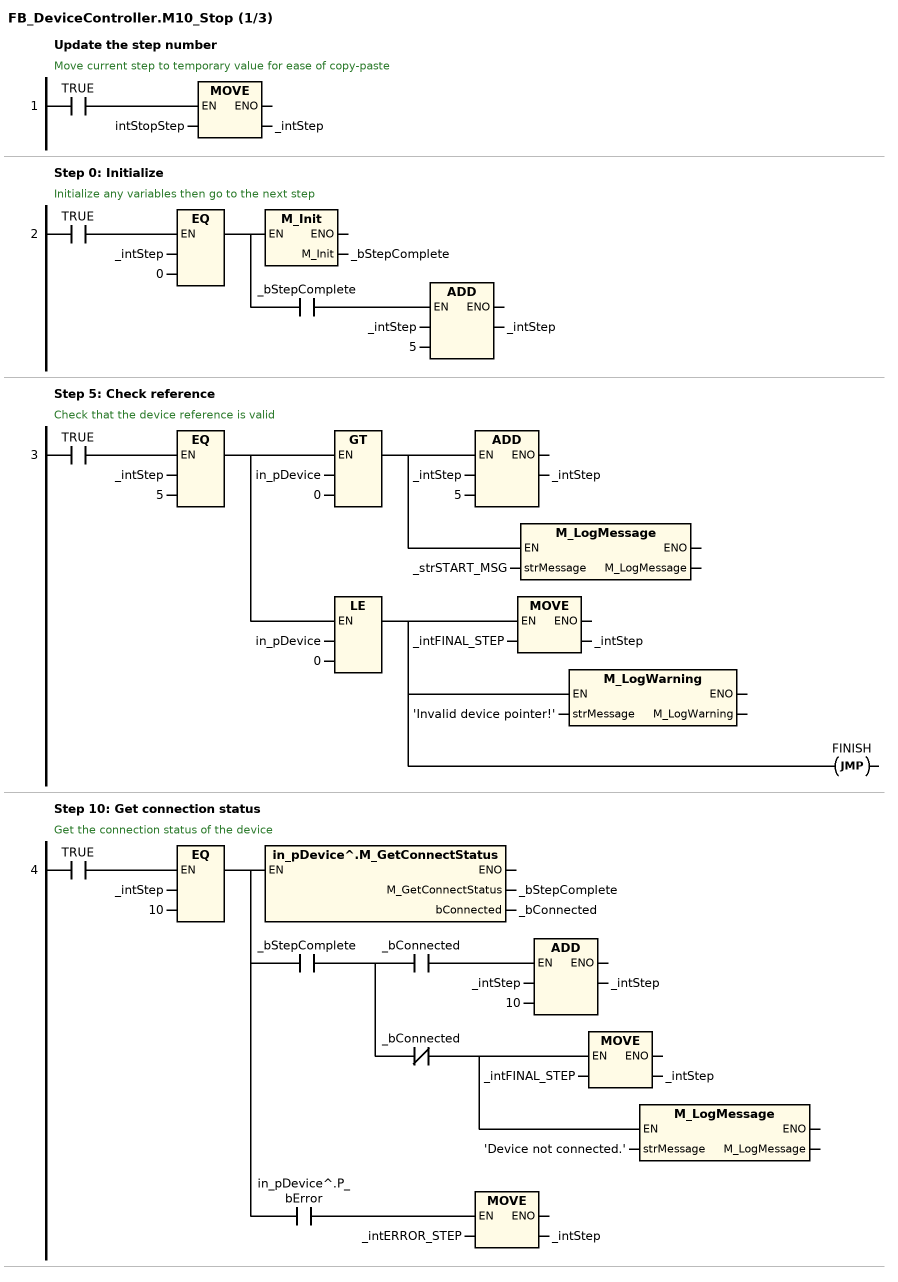
// NETWORK 1: Update the step number
// Move current step to temporary value for ease of copy-paste
_intStep := intStopStep;

// NETWORK 2: Step 0: Initialize
// Initialize any variables then go to the next step
_w1 := _intStep = 0;
IF _w1 THEN _bStepComplete := M_Init(); END_IF
IF _w1 AND _bStepComplete THEN _intStep := _intStep + 5; END_IF

// NETWORK 3: Step 5: Check reference
// Check that the device reference is valid
_w2 := _intStep = 5;
_w3 := _w2 AND in_pDevice > 0;
IF _w3 THEN _intStep := _intStep + 5; END_IF
IF _w3 THEN M_LogMessage(strMessage := _strSTART_MSG); END_IF
_w4 := _w2 AND in_pDevice <= 0;
IF _w4 THEN _intStep := _intFINAL_STEP; END_IF
IF _w4 THEN M_LogWarning(strMessage := 'Invalid device pointer!'); END_IF
IF _w4 THEN JMP FINISH; END_IF

// NETWORK 4: Step 10: Get connection status
// Get the connection status of the device
_w5 := _intStep = 10;
IF _w5 THEN _bStepComplete := in_pDevice^.M_GetConnectStatus(bConnected => _bConnected); END_IF
_w6 := _w5 AND _bStepComplete;
IF _w6 AND _bConnected THEN _intStep := _intStep + 10; END_IF
_w7 := _w6 AND NOT _bConnected;
IF _w7 THEN _intStep := _intFINAL_STEP; END_IF
IF _w7 THEN M_LogMessage(strMessage := 'Device not connected.'); END_IF
IF _w5 AND in_pDevice^.P_bError THEN _intStep := _intERROR_STEP; END_IF

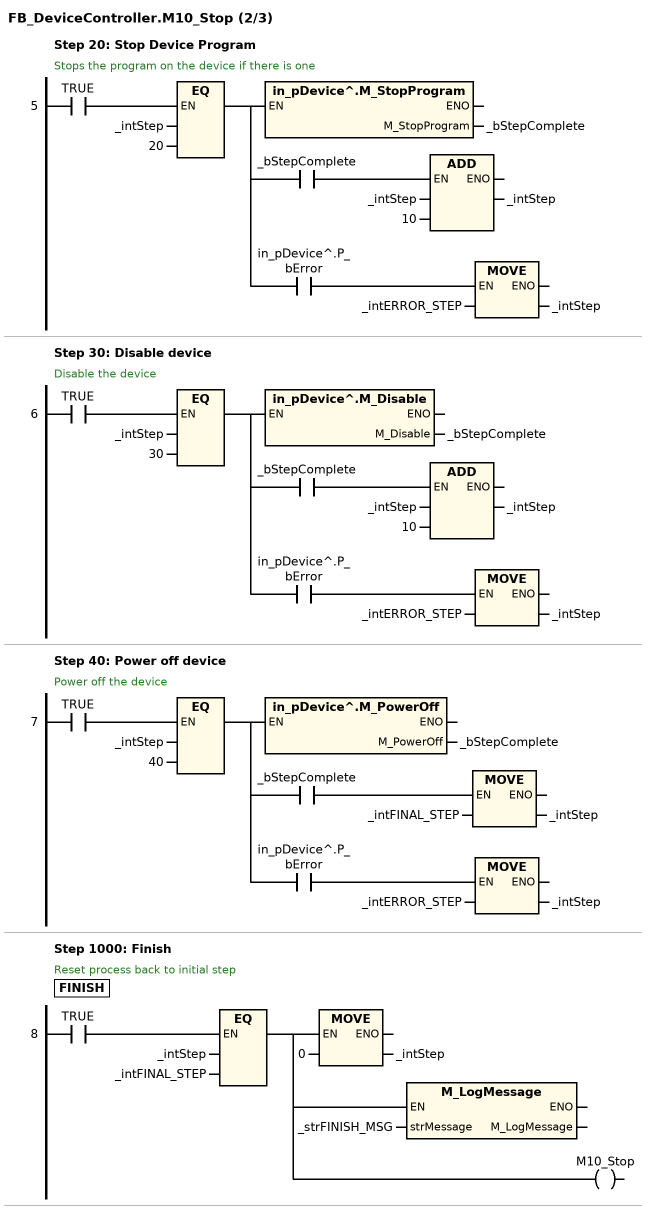
// NETWORK 5: Step 20: Stop Device Program
// Stops the program on the device if there is one
_w8 := _intStep = 20;
IF _w8 THEN _bStepComplete := in_pDevice^.M_StopProgram(); END_IF
IF _w8 AND _bStepComplete THEN _intStep := _intStep + 10; END_IF
IF _w8 AND in_pDevice^.P_bError THEN _intStep := _intERROR_STEP; END_IF

// NETWORK 6: Step 30: Disable device
// Disable the device
_w9 := _intStep = 30;
IF _w9 THEN _bStepComplete := in_pDevice^.M_Disable(); END_IF
IF _w9 AND _bStepComplete THEN _intStep := _intStep + 10; END_IF
IF _w9 AND in_pDevice^.P_bError THEN _intStep := _intERROR_STEP; END_IF

// NETWORK 7: Step 40: Power off device
// Power off the device
_w10 := _intStep = 40;
IF _w10 THEN _bStepComplete := in_pDevice^.M_PowerOff(); END_IF
IF _w10 AND _bStepComplete THEN _intStep := _intFINAL_STEP; END_IF
IF _w10 AND in_pDevice^.P_bError THEN _intStep := _intERROR_STEP; END_IF

// NETWORK 8: Step 1000: Finish
// Reset process back to initial step
FINISH:
_w11 := _intStep = _intFINAL_STEP;
IF _w11 THEN _intStep := 0; END_IF
IF _w11 THEN M_LogMessage(strMessage := _strFINISH_MSG); END_IF
M10_Stop := _w11;

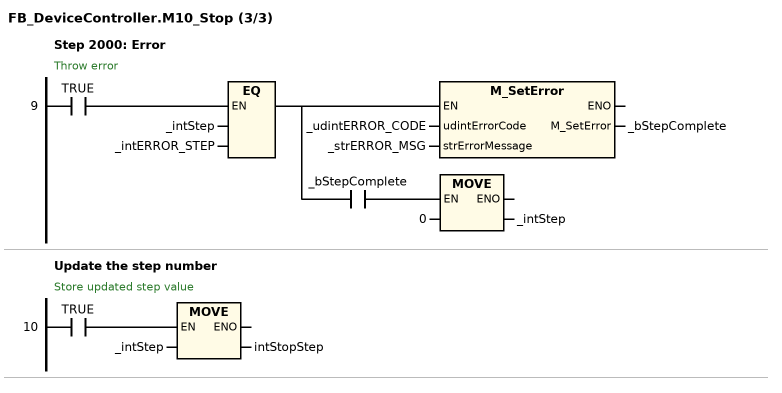
// NETWORK 9: Step 2000: Error
// Throw error
_w12 := _intStep = _intERROR_STEP;
IF _w12 THEN
    _bStepComplete := M_SetError(udintErrorCode := _udintERROR_CODE, strErrorMessage := _strERROR_MSG);
END_IF
IF _w12 AND _bStepComplete THEN _intStep := 0; END_IF

// NETWORK 10: Update the step number
// Store updated step value
intStopStep := _intStep;
END_METHOD

(* Connects, resets, and powers on the device. *)
METHOD M20_Reset : BOOL
VAR CONSTANT
	_intFINAL_STEP : INT := 1000;
	_intERROR_STEP : INT := 2000;
	_udintERROR_CODE: UDINT := E_DeviceControllerError.ResetError;
	_strERROR_MSG: T_MaxString := 'Error while trying to reset device!';
	_strSTART_MSG: T_MaxString := 'Resetting device';
	_strFINISH_MSG: T_MaxString := 'Device reset';
END_VAR
VAR
	_bStepComplete: BOOL;
	_intStep: INT;
END_VAR
VAR_INST // added by the converter: edge detectors and wires of the graphical bodies
    _w1, _w2, _w3, _w4, _w5, _w6, _w7, _w8, _w9 : BOOL;
END_VAR
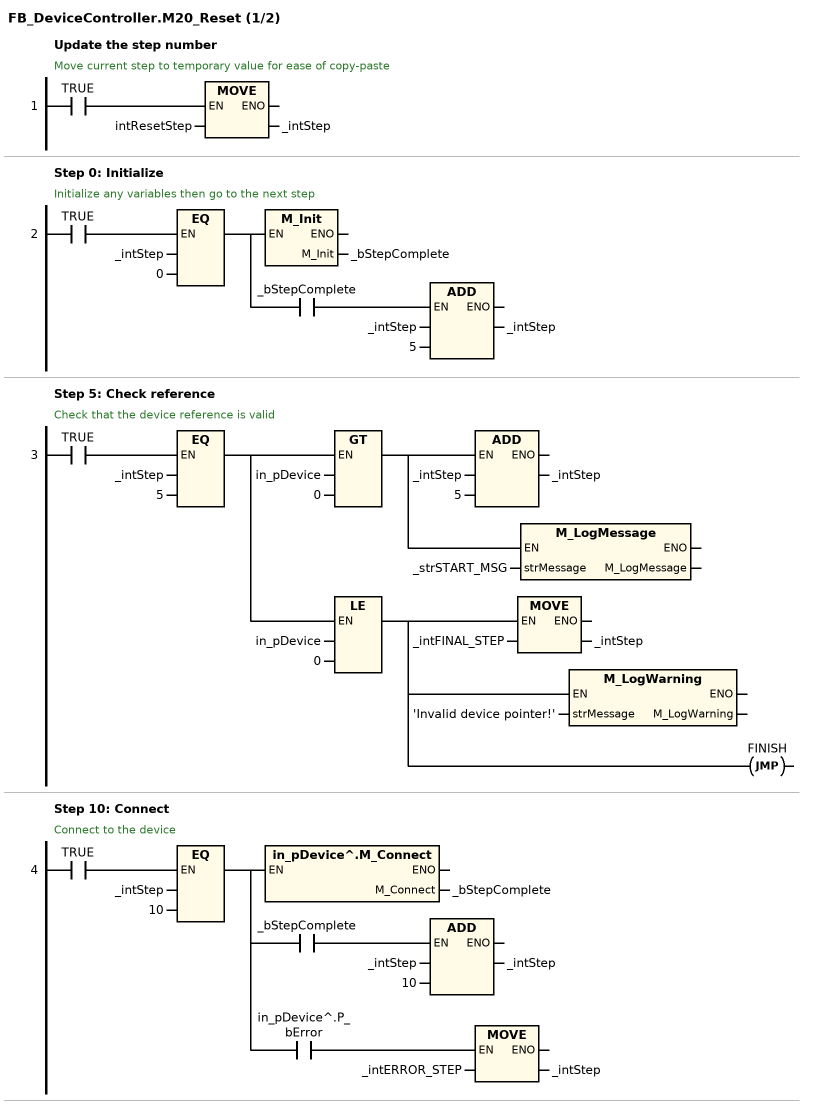
// NETWORK 1: Update the step number
// Move current step to temporary value for ease of copy-paste
_intStep := intResetStep;

// NETWORK 2: Step 0: Initialize
// Initialize any variables then go to the next step
_w1 := _intStep = 0;
IF _w1 THEN _bStepComplete := M_Init(); END_IF
IF _w1 AND _bStepComplete THEN _intStep := _intStep + 5; END_IF

// NETWORK 3: Step 5: Check reference
// Check that the device reference is valid
_w2 := _intStep = 5;
_w3 := _w2 AND in_pDevice > 0;
IF _w3 THEN _intStep := _intStep + 5; END_IF
IF _w3 THEN M_LogMessage(strMessage := _strSTART_MSG); END_IF
_w4 := _w2 AND in_pDevice <= 0;
IF _w4 THEN _intStep := _intFINAL_STEP; END_IF
IF _w4 THEN M_LogWarning(strMessage := 'Invalid device pointer!'); END_IF
IF _w4 THEN JMP FINISH; END_IF

// NETWORK 4: Step 10: Connect
// Connect to the device
_w5 := _intStep = 10;
IF _w5 THEN _bStepComplete := in_pDevice^.M_Connect(); END_IF
IF _w5 AND _bStepComplete THEN _intStep := _intStep + 10; END_IF
IF _w5 AND in_pDevice^.P_bError THEN _intStep := _intERROR_STEP; END_IF

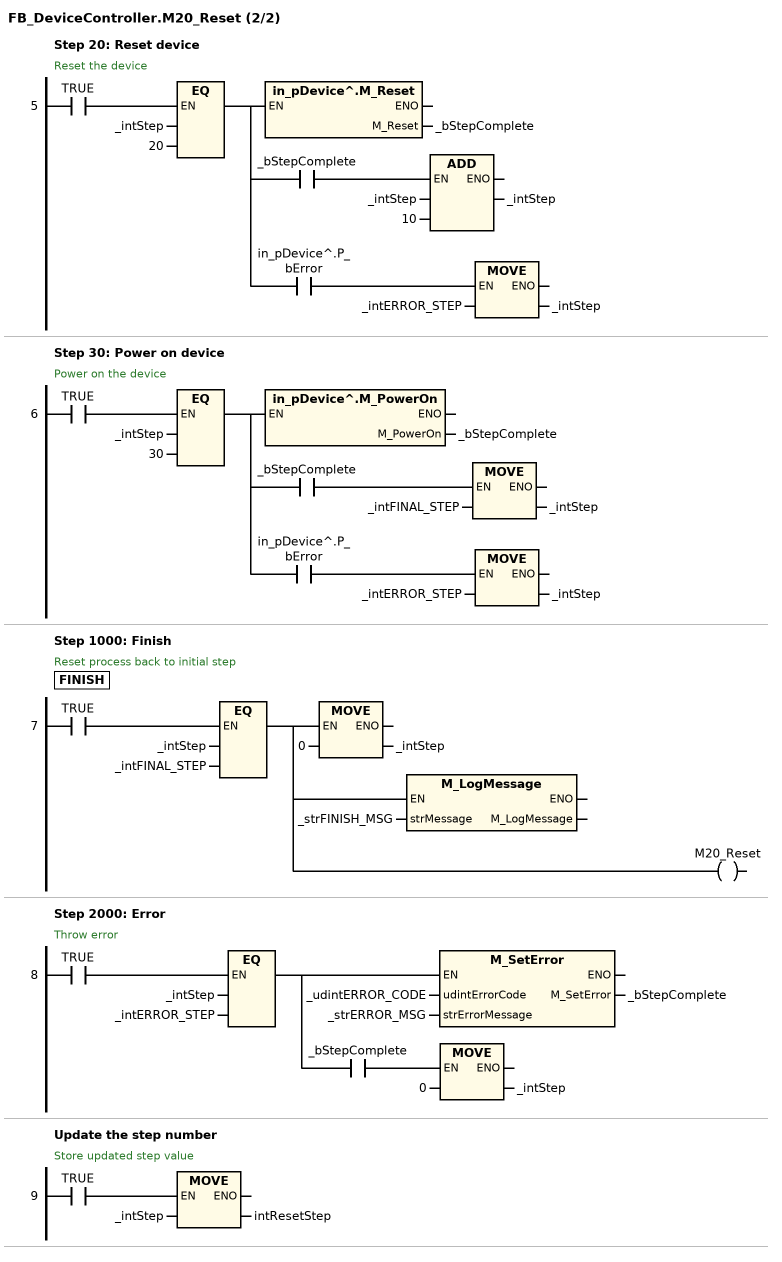
// NETWORK 5: Step 20: Reset device
// Reset the device
_w6 := _intStep = 20;
IF _w6 THEN _bStepComplete := in_pDevice^.M_Reset(); END_IF
IF _w6 AND _bStepComplete THEN _intStep := _intStep + 10; END_IF
IF _w6 AND in_pDevice^.P_bError THEN _intStep := _intERROR_STEP; END_IF

// NETWORK 6: Step 30: Power on device
// Power on the device
_w7 := _intStep = 30;
IF _w7 THEN _bStepComplete := in_pDevice^.M_PowerOn(); END_IF
IF _w7 AND _bStepComplete THEN _intStep := _intFINAL_STEP; END_IF
IF _w7 AND in_pDevice^.P_bError THEN _intStep := _intERROR_STEP; END_IF

// NETWORK 7: Step 1000: Finish
// Reset process back to initial step
FINISH:
_w8 := _intStep = _intFINAL_STEP;
IF _w8 THEN _intStep := 0; END_IF
IF _w8 THEN M_LogMessage(strMessage := _strFINISH_MSG); END_IF
M20_Reset := _w8;

// NETWORK 8: Step 2000: Error
// Throw error
_w9 := _intStep = _intERROR_STEP;
IF _w9 THEN
    _bStepComplete := M_SetError(udintErrorCode := _udintERROR_CODE, strErrorMessage := _strERROR_MSG);
END_IF
IF _w9 AND _bStepComplete THEN _intStep := 0; END_IF

// NETWORK 9: Update the step number
// Store updated step value
intResetStep := _intStep;
END_METHOD

(* Loads program and starts device then returns TRUE. *)
METHOD M30_Start : BOOL
VAR CONSTANT
	_udintERROR_CODE: UDINT := E_DeviceControllerError.StartError;
	_strERROR_MSG: T_MaxString := 'Error while trying to start device!';
	_intFINAL_STEP : INT := 1000;
	_intERROR_STEP : INT := 2000;
	_strSTART_MSG: T_MaxString := 'Starting device';
	_strFINISH_MSG: T_MaxString := 'Device started';
END_VAR
VAR
	_bStepComplete: BOOL;
	_intStep: INT;
END_VAR
VAR_INST // added by the converter: edge detectors and wires of the graphical bodies
    _w1, _w2, _w3, _w4, _w5, _w6, _w7, _w8, _w9 : BOOL;
END_VAR
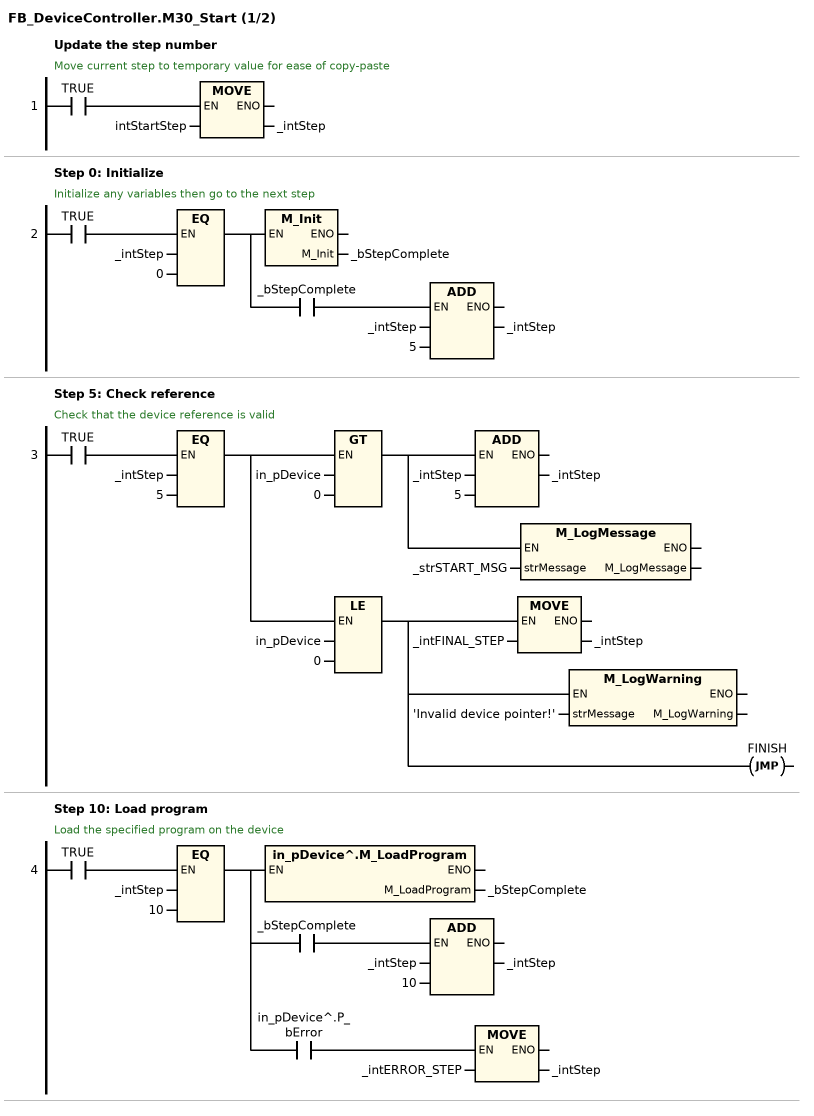
// NETWORK 1: Update the step number
// Move current step to temporary value for ease of copy-paste
_intStep := intStartStep;

// NETWORK 2: Step 0: Initialize
// Initialize any variables then go to the next step
_w1 := _intStep = 0;
IF _w1 THEN _bStepComplete := M_Init(); END_IF
IF _w1 AND _bStepComplete THEN _intStep := _intStep + 5; END_IF

// NETWORK 3: Step 5: Check reference
// Check that the device reference is valid
_w2 := _intStep = 5;
_w3 := _w2 AND in_pDevice > 0;
IF _w3 THEN _intStep := _intStep + 5; END_IF
IF _w3 THEN M_LogMessage(strMessage := _strSTART_MSG); END_IF
_w4 := _w2 AND in_pDevice <= 0;
IF _w4 THEN _intStep := _intFINAL_STEP; END_IF
IF _w4 THEN M_LogWarning(strMessage := 'Invalid device pointer!'); END_IF
IF _w4 THEN JMP FINISH; END_IF

// NETWORK 4: Step 10: Load program
// Load the specified program on the device
_w5 := _intStep = 10;
IF _w5 THEN _bStepComplete := in_pDevice^.M_LoadProgram(); END_IF
IF _w5 AND _bStepComplete THEN _intStep := _intStep + 10; END_IF
IF _w5 AND in_pDevice^.P_bError THEN _intStep := _intERROR_STEP; END_IF

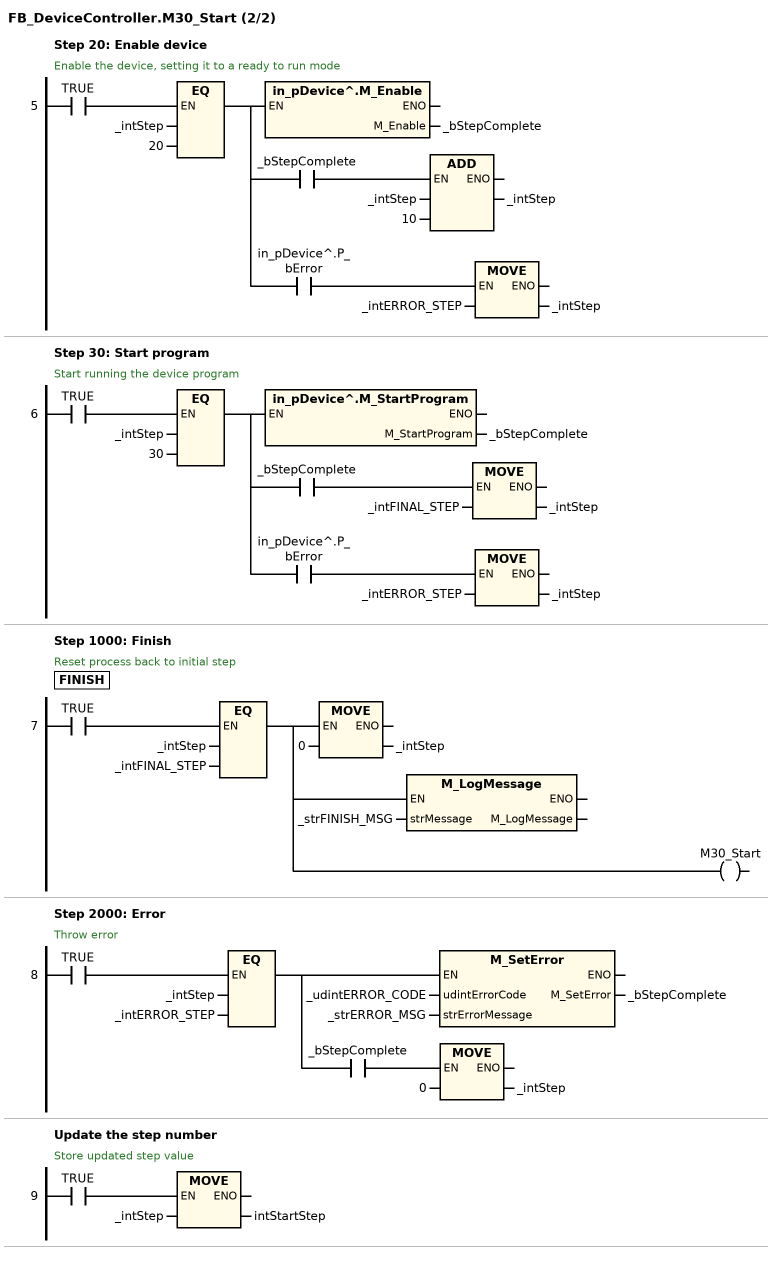
// NETWORK 5: Step 20: Enable device
// Enable the device, setting it to a ready to run mode
_w6 := _intStep = 20;
IF _w6 THEN _bStepComplete := in_pDevice^.M_Enable(); END_IF
IF _w6 AND _bStepComplete THEN _intStep := _intStep + 10; END_IF
IF _w6 AND in_pDevice^.P_bError THEN _intStep := _intERROR_STEP; END_IF

// NETWORK 6: Step 30: Start program
// Start running the device program
_w7 := _intStep = 30;
IF _w7 THEN _bStepComplete := in_pDevice^.M_StartProgram(); END_IF
IF _w7 AND _bStepComplete THEN _intStep := _intFINAL_STEP; END_IF
IF _w7 AND in_pDevice^.P_bError THEN _intStep := _intERROR_STEP; END_IF

// NETWORK 7: Step 1000: Finish
// Reset process back to initial step
FINISH:
_w8 := _intStep = _intFINAL_STEP;
IF _w8 THEN _intStep := 0; END_IF
IF _w8 THEN M_LogMessage(strMessage := _strFINISH_MSG); END_IF
M30_Start := _w8;

// NETWORK 8: Step 2000: Error
// Throw error
_w9 := _intStep = _intERROR_STEP;
IF _w9 THEN
    _bStepComplete := M_SetError(udintErrorCode := _udintERROR_CODE, strErrorMessage := _strERROR_MSG);
END_IF
IF _w9 AND _bStepComplete THEN _intStep := 0; END_IF

// NETWORK 9: Update the step number
// Store updated step value
intStartStep := _intStep;
END_METHOD

(* Stops and disables the device then returns TRUE when done. *)
METHOD M32_Complete : BOOL
VAR CONSTANT
	_udintERROR_CODE: UDINT := E_DeviceControllerError.CompleteError;
	_strERROR_MSG: T_MaxString := 'Error while trying to complete device!';
	_intFINAL_STEP : INT := 1000;
	_intERROR_STEP : INT := 2000;
	_strSTART_MSG: T_MaxString := 'Completing device';
	_strFINISH_MSG: T_MaxString := 'Device completed';
END_VAR
VAR
	_bStepComplete: BOOL;
	_intStep: INT;
END_VAR
VAR_INST // added by the converter: edge detectors and wires of the graphical bodies
    _w1, _w2, _w3, _w4, _w5, _w6, _w7, _w8 : BOOL;
END_VAR
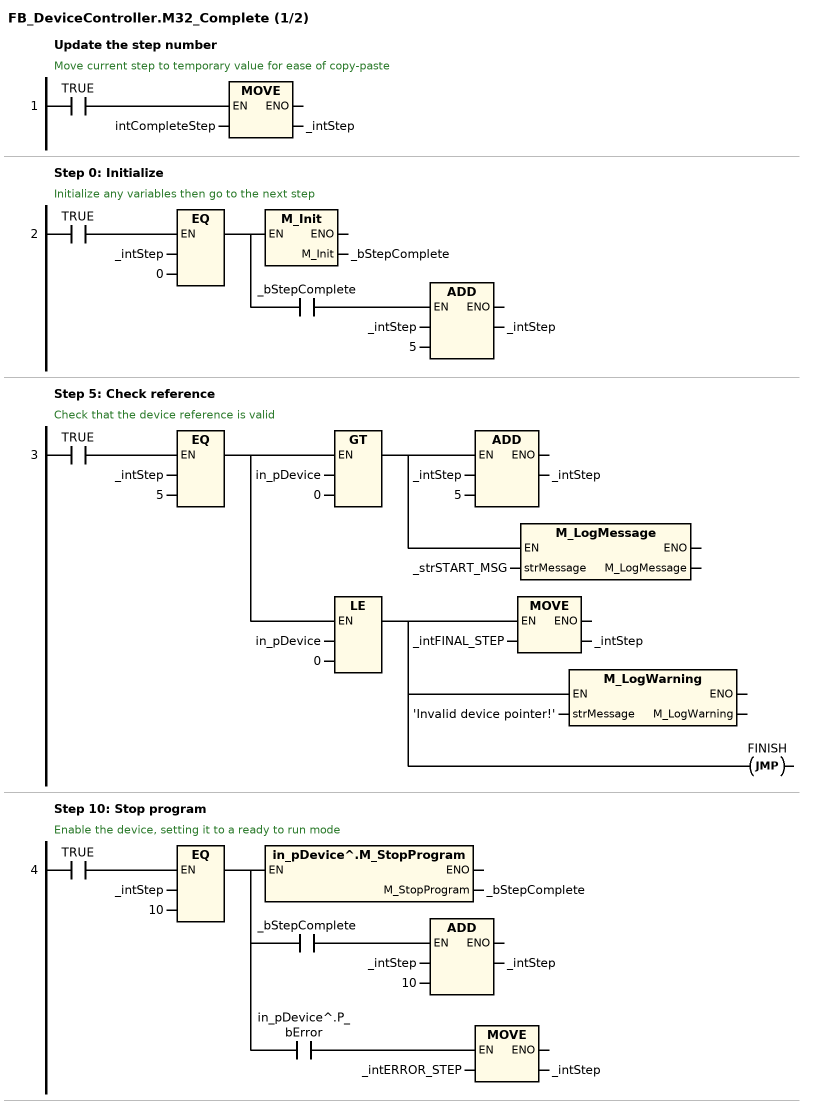
// NETWORK 1: Update the step number
// Move current step to temporary value for ease of copy-paste
_intStep := intCompleteStep;

// NETWORK 2: Step 0: Initialize
// Initialize any variables then go to the next step
_w1 := _intStep = 0;
IF _w1 THEN _bStepComplete := M_Init(); END_IF
IF _w1 AND _bStepComplete THEN _intStep := _intStep + 5; END_IF

// NETWORK 3: Step 5: Check reference
// Check that the device reference is valid
_w2 := _intStep = 5;
_w3 := _w2 AND in_pDevice > 0;
IF _w3 THEN _intStep := _intStep + 5; END_IF
IF _w3 THEN M_LogMessage(strMessage := _strSTART_MSG); END_IF
_w4 := _w2 AND in_pDevice <= 0;
IF _w4 THEN _intStep := _intFINAL_STEP; END_IF
IF _w4 THEN M_LogWarning(strMessage := 'Invalid device pointer!'); END_IF
IF _w4 THEN JMP FINISH; END_IF

// NETWORK 4: Step 10: Stop program
// Enable the device, setting it to a ready to run mode
_w5 := _intStep = 10;
IF _w5 THEN _bStepComplete := in_pDevice^.M_StopProgram(); END_IF
IF _w5 AND _bStepComplete THEN _intStep := _intStep + 10; END_IF
IF _w5 AND in_pDevice^.P_bError THEN _intStep := _intERROR_STEP; END_IF

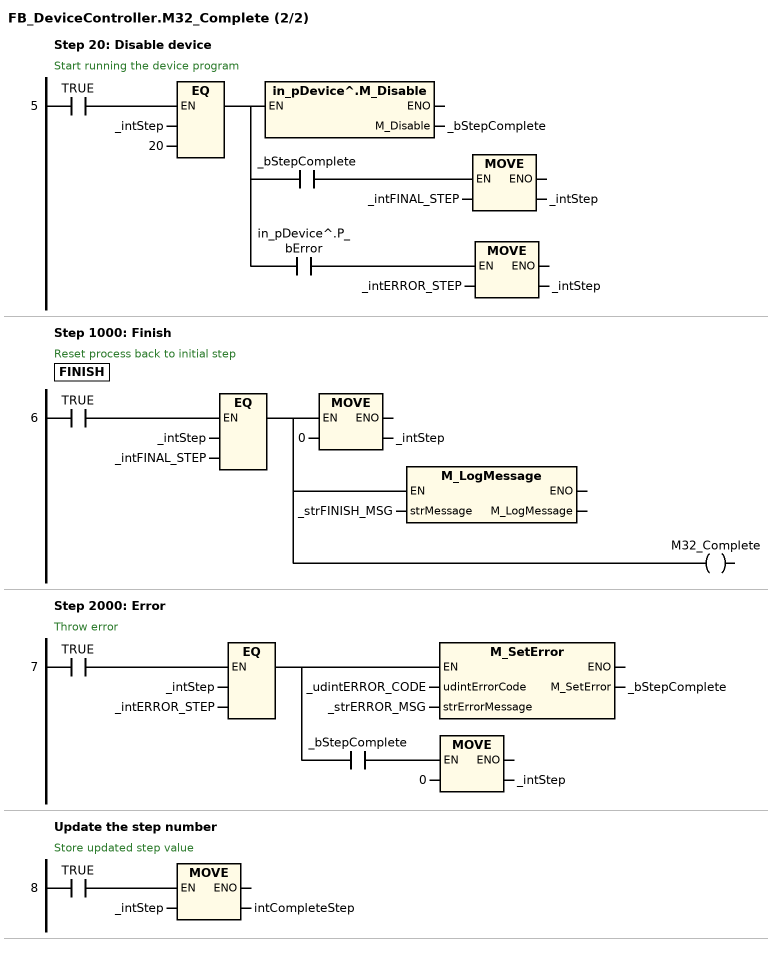
// NETWORK 5: Step 20: Disable device
// Start running the device program
_w6 := _intStep = 20;
IF _w6 THEN _bStepComplete := in_pDevice^.M_Disable(); END_IF
IF _w6 AND _bStepComplete THEN _intStep := _intFINAL_STEP; END_IF
IF _w6 AND in_pDevice^.P_bError THEN _intStep := _intERROR_STEP; END_IF

// NETWORK 6: Step 1000: Finish
// Reset process back to initial step
FINISH:
_w7 := _intStep = _intFINAL_STEP;
IF _w7 THEN _intStep := 0; END_IF
IF _w7 THEN M_LogMessage(strMessage := _strFINISH_MSG); END_IF
M32_Complete := _w7;

// NETWORK 7: Step 2000: Error
// Throw error
_w8 := _intStep = _intERROR_STEP;
IF _w8 THEN
    _bStepComplete := M_SetError(udintErrorCode := _udintERROR_CODE, strErrorMessage := _strERROR_MSG);
END_IF
IF _w8 AND _bStepComplete THEN _intStep := 0; END_IF

// NETWORK 8: Update the step number
// Store updated step value
intCompleteStep := _intStep;
END_METHOD

(* Pauses the device then returns TRUE. *)
METHOD M40_Hold : BOOL
VAR CONSTANT
	_udintERROR_CODE: UDINT := E_DeviceControllerError.HoldError;
	_strERROR_MSG: T_MaxString := 'Error while trying to hold device!';
	_intFINAL_STEP : INT := 1000;
	_intERROR_STEP : INT := 2000;
	_strSTART_MSG: T_MaxString := 'Holding device';
	_strFINISH_MSG: T_MaxString := 'Device held';
END_VAR
VAR
	_bStepComplete: BOOL;
	_intStep: INT;
END_VAR
VAR_INST // added by the converter: edge detectors and wires of the graphical bodies
    _w1, _w2, _w3, _w4, _w5, _w6, _w7 : BOOL;
END_VAR
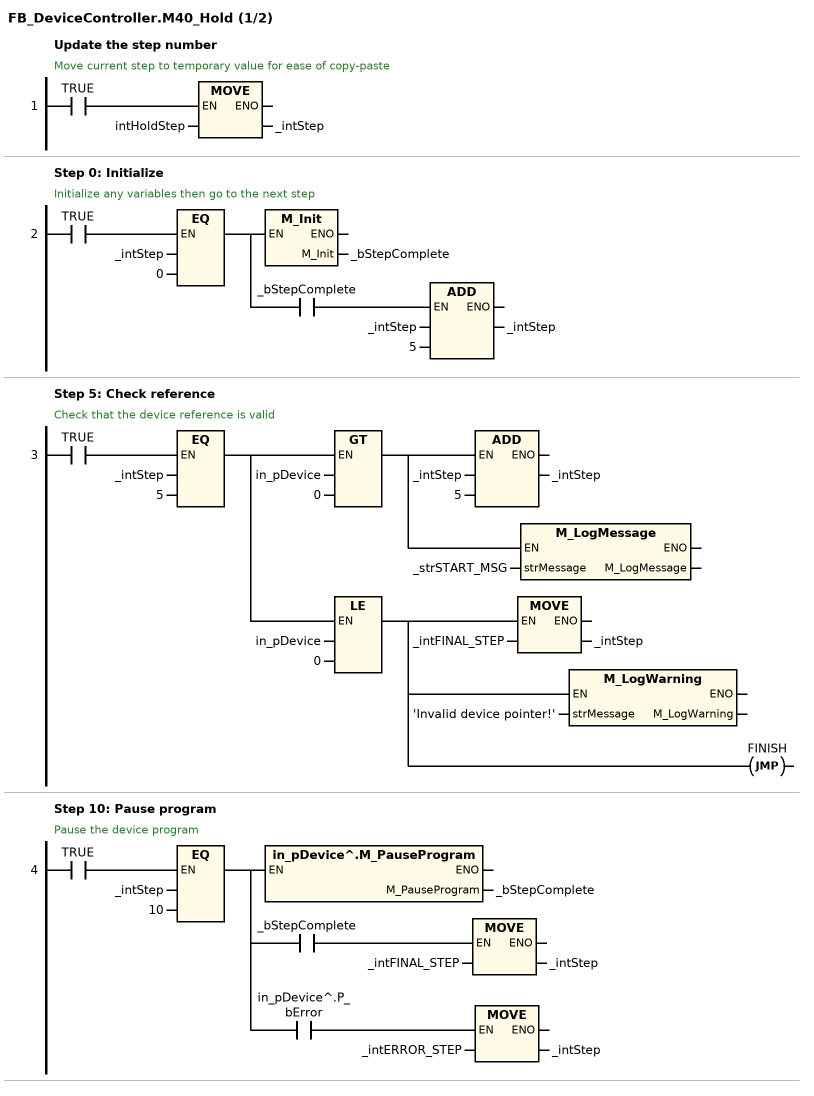
// NETWORK 1: Update the step number
// Move current step to temporary value for ease of copy-paste
_intStep := intHoldStep;

// NETWORK 2: Step 0: Initialize
// Initialize any variables then go to the next step
_w1 := _intStep = 0;
IF _w1 THEN _bStepComplete := M_Init(); END_IF
IF _w1 AND _bStepComplete THEN _intStep := _intStep + 5; END_IF

// NETWORK 3: Step 5: Check reference
// Check that the device reference is valid
_w2 := _intStep = 5;
_w3 := _w2 AND in_pDevice > 0;
IF _w3 THEN _intStep := _intStep + 5; END_IF
IF _w3 THEN M_LogMessage(strMessage := _strSTART_MSG); END_IF
_w4 := _w2 AND in_pDevice <= 0;
IF _w4 THEN _intStep := _intFINAL_STEP; END_IF
IF _w4 THEN M_LogWarning(strMessage := 'Invalid device pointer!'); END_IF
IF _w4 THEN JMP FINISH; END_IF

// NETWORK 4: Step 10: Pause program
// Pause the device program
_w5 := _intStep = 10;
IF _w5 THEN _bStepComplete := in_pDevice^.M_PauseProgram(); END_IF
IF _w5 AND _bStepComplete THEN _intStep := _intFINAL_STEP; END_IF
IF _w5 AND in_pDevice^.P_bError THEN _intStep := _intERROR_STEP; END_IF

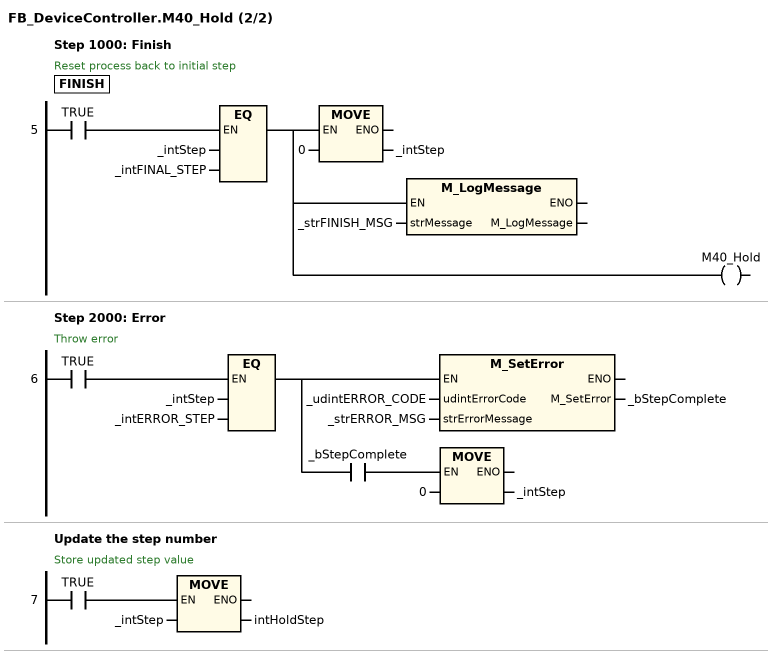
// NETWORK 5: Step 1000: Finish
// Reset process back to initial step
FINISH:
_w6 := _intStep = _intFINAL_STEP;
IF _w6 THEN _intStep := 0; END_IF
IF _w6 THEN M_LogMessage(strMessage := _strFINISH_MSG); END_IF
M40_Hold := _w6;

// NETWORK 6: Step 2000: Error
// Throw error
_w7 := _intStep = _intERROR_STEP;
IF _w7 THEN
    _bStepComplete := M_SetError(udintErrorCode := _udintERROR_CODE, strErrorMessage := _strERROR_MSG);
END_IF
IF _w7 AND _bStepComplete THEN _intStep := 0; END_IF

// NETWORK 7: Update the step number
// Store updated step value
intHoldStep := _intStep;
END_METHOD

(* Unpauses the device then returns TRUE. *)
METHOD M42_Unhold : BOOL
VAR CONSTANT
	_udintERROR_CODE: UDINT := E_DeviceControllerError.UnholdError;
	_strERROR_MSG: T_MaxString := 'Error while trying to unhold device!';
	_intFINAL_STEP : INT := 1000;
	_intERROR_STEP : INT := 2000;
	_strSTART_MSG: T_MaxString := 'Unholding device';
	_strFINISH_MSG: T_MaxString := 'Device unheld';
END_VAR
VAR
	_bStepComplete: BOOL;
	_intStep: INT;
END_VAR
VAR_INST // added by the converter: edge detectors and wires of the graphical bodies
    _w1, _w2, _w3, _w4, _w5, _w6, _w7 : BOOL;
END_VAR
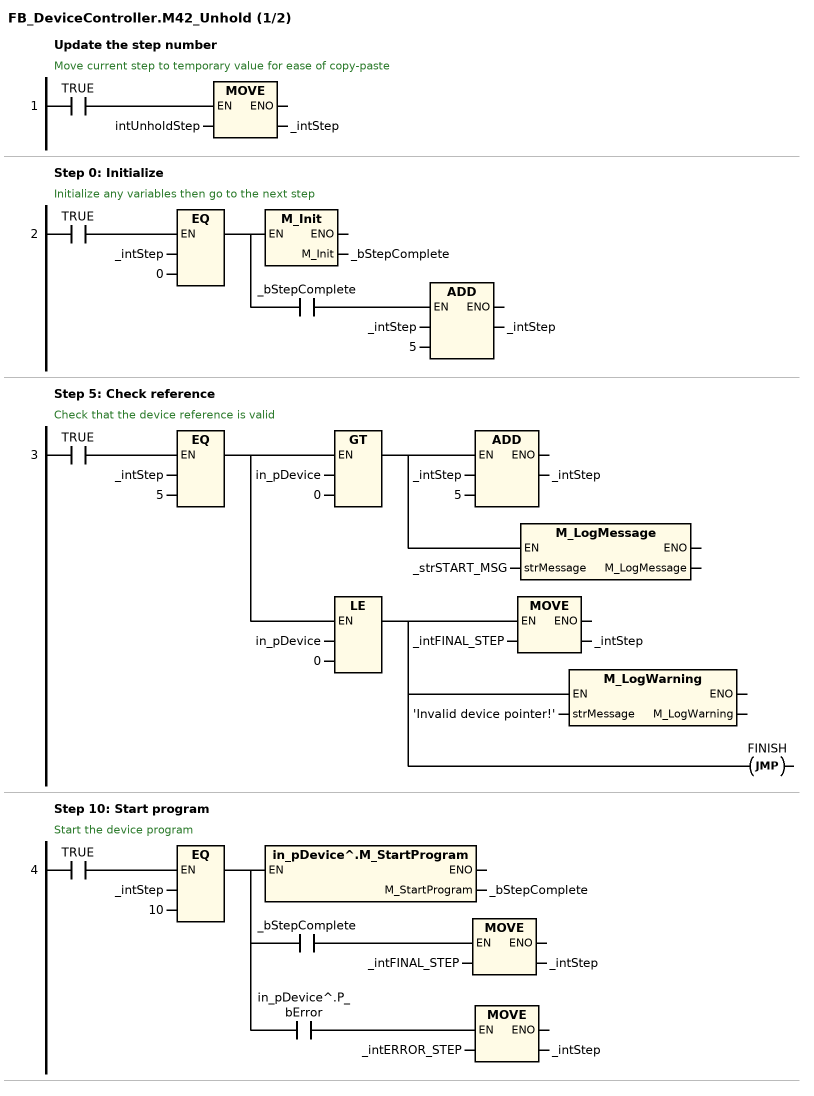
// NETWORK 1: Update the step number
// Move current step to temporary value for ease of copy-paste
_intStep := intUnholdStep;

// NETWORK 2: Step 0: Initialize
// Initialize any variables then go to the next step
_w1 := _intStep = 0;
IF _w1 THEN _bStepComplete := M_Init(); END_IF
IF _w1 AND _bStepComplete THEN _intStep := _intStep + 5; END_IF

// NETWORK 3: Step 5: Check reference
// Check that the device reference is valid
_w2 := _intStep = 5;
_w3 := _w2 AND in_pDevice > 0;
IF _w3 THEN _intStep := _intStep + 5; END_IF
IF _w3 THEN M_LogMessage(strMessage := _strSTART_MSG); END_IF
_w4 := _w2 AND in_pDevice <= 0;
IF _w4 THEN _intStep := _intFINAL_STEP; END_IF
IF _w4 THEN M_LogWarning(strMessage := 'Invalid device pointer!'); END_IF
IF _w4 THEN JMP FINISH; END_IF

// NETWORK 4: Step 10: Start program
// Start the device program
_w5 := _intStep = 10;
IF _w5 THEN _bStepComplete := in_pDevice^.M_StartProgram(); END_IF
IF _w5 AND _bStepComplete THEN _intStep := _intFINAL_STEP; END_IF
IF _w5 AND in_pDevice^.P_bError THEN _intStep := _intERROR_STEP; END_IF

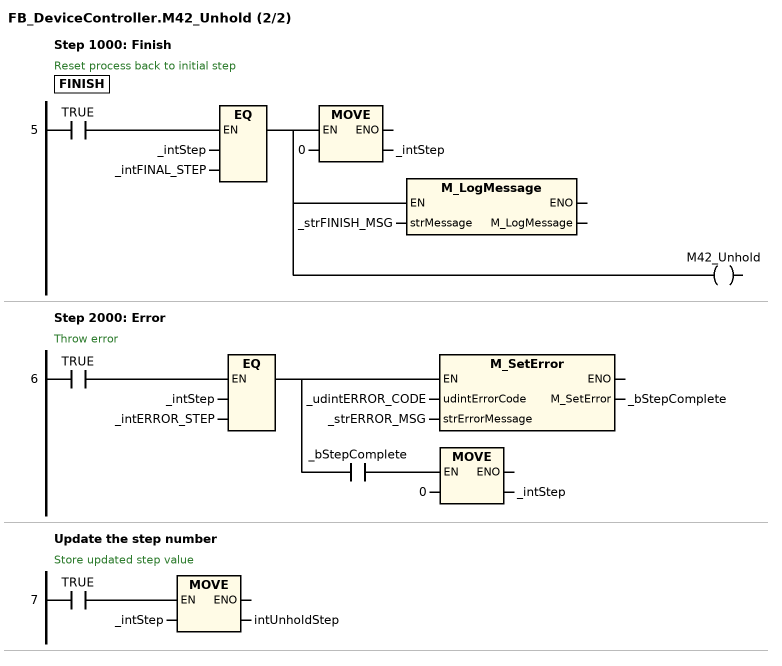
// NETWORK 5: Step 1000: Finish
// Reset process back to initial step
FINISH:
_w6 := _intStep = _intFINAL_STEP;
IF _w6 THEN _intStep := 0; END_IF
IF _w6 THEN M_LogMessage(strMessage := _strFINISH_MSG); END_IF
M42_Unhold := _w6;

// NETWORK 6: Step 2000: Error
// Throw error
_w7 := _intStep = _intERROR_STEP;
IF _w7 THEN
    _bStepComplete := M_SetError(udintErrorCode := _udintERROR_CODE, strErrorMessage := _strERROR_MSG);
END_IF
IF _w7 AND _bStepComplete THEN _intStep := 0; END_IF

// NETWORK 7: Update the step number
// Store updated step value
intUnholdStep := _intStep;
END_METHOD

(* Pauses the device then returns TRUE. *)
METHOD M50_Suspend : BOOL
VAR CONSTANT
	_udintERROR_CODE: UDINT := E_DeviceControllerError.SuspendError;
	_strERROR_MSG: T_MaxString := 'Error while trying to suspend device!';
	_intFINAL_STEP : INT := 1000;
	_intERROR_STEP : INT := 2000;
	_strSTART_MSG: T_MaxString := 'Suspending device';
	_strFINISH_MSG: T_MaxString := 'Device suspended';
END_VAR
VAR
	_bStepComplete: BOOL;
	_intStep: INT;
END_VAR
VAR_INST // added by the converter: edge detectors and wires of the graphical bodies
    _w1, _w2, _w3, _w4, _w5, _w6, _w7 : BOOL;
END_VAR
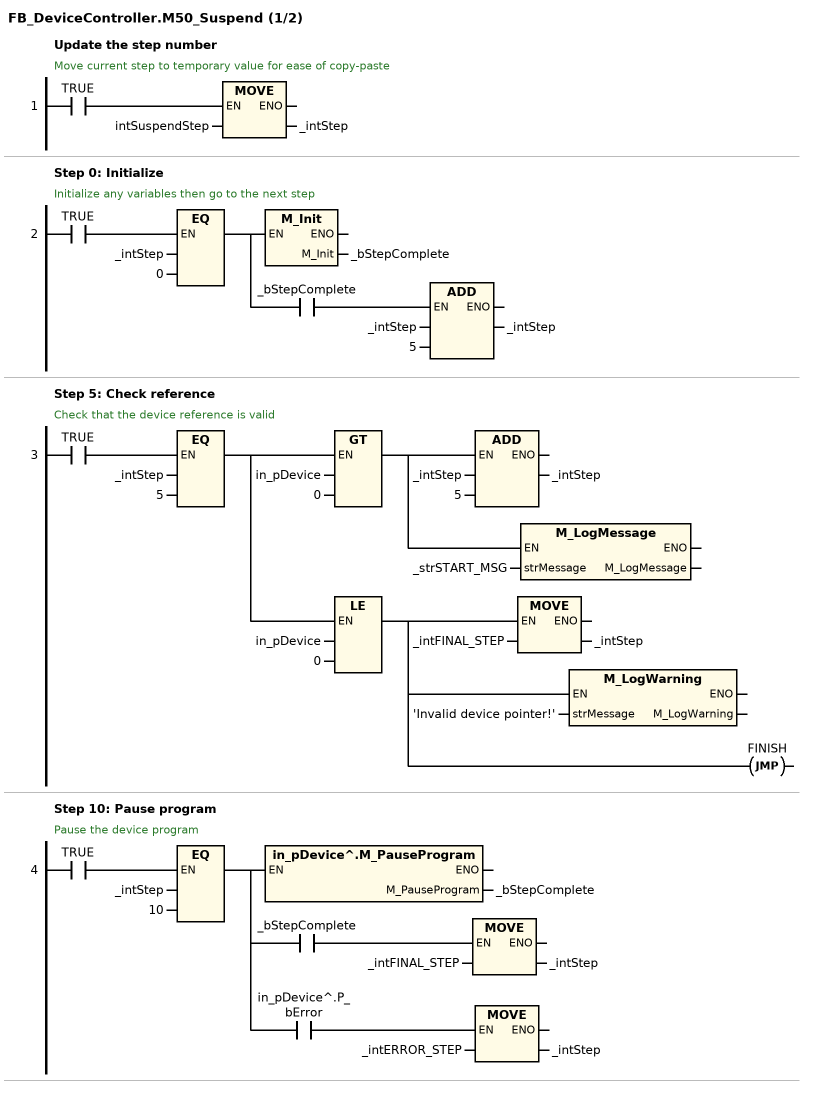
// NETWORK 1: Update the step number
// Move current step to temporary value for ease of copy-paste
_intStep := intSuspendStep;

// NETWORK 2: Step 0: Initialize
// Initialize any variables then go to the next step
_w1 := _intStep = 0;
IF _w1 THEN _bStepComplete := M_Init(); END_IF
IF _w1 AND _bStepComplete THEN _intStep := _intStep + 5; END_IF

// NETWORK 3: Step 5: Check reference
// Check that the device reference is valid
_w2 := _intStep = 5;
_w3 := _w2 AND in_pDevice > 0;
IF _w3 THEN _intStep := _intStep + 5; END_IF
IF _w3 THEN M_LogMessage(strMessage := _strSTART_MSG); END_IF
_w4 := _w2 AND in_pDevice <= 0;
IF _w4 THEN _intStep := _intFINAL_STEP; END_IF
IF _w4 THEN M_LogWarning(strMessage := 'Invalid device pointer!'); END_IF
IF _w4 THEN JMP FINISH; END_IF

// NETWORK 4: Step 10: Pause program
// Pause the device program
_w5 := _intStep = 10;
IF _w5 THEN _bStepComplete := in_pDevice^.M_PauseProgram(); END_IF
IF _w5 AND _bStepComplete THEN _intStep := _intFINAL_STEP; END_IF
IF _w5 AND in_pDevice^.P_bError THEN _intStep := _intERROR_STEP; END_IF

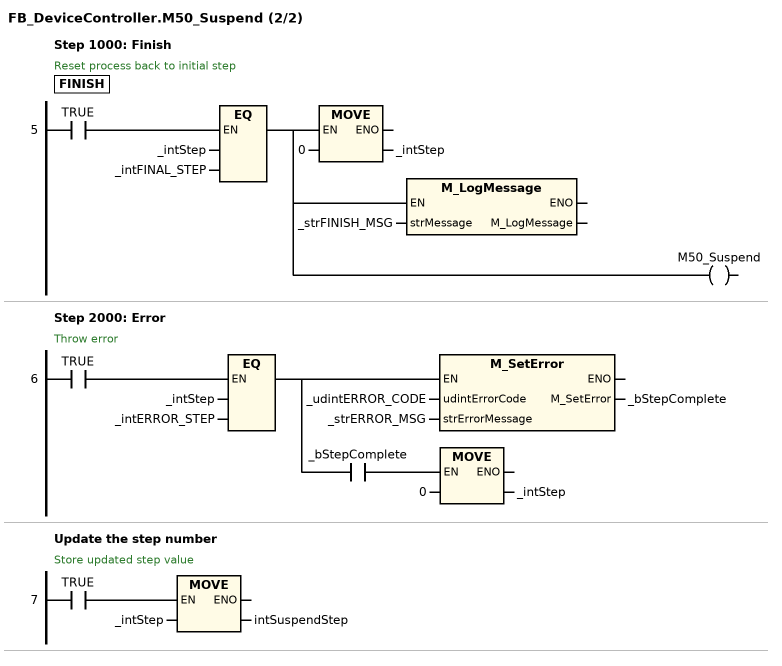
// NETWORK 5: Step 1000: Finish
// Reset process back to initial step
FINISH:
_w6 := _intStep = _intFINAL_STEP;
IF _w6 THEN _intStep := 0; END_IF
IF _w6 THEN M_LogMessage(strMessage := _strFINISH_MSG); END_IF
M50_Suspend := _w6;

// NETWORK 6: Step 2000: Error
// Throw error
_w7 := _intStep = _intERROR_STEP;
IF _w7 THEN
    _bStepComplete := M_SetError(udintErrorCode := _udintERROR_CODE, strErrorMessage := _strERROR_MSG);
END_IF
IF _w7 AND _bStepComplete THEN _intStep := 0; END_IF

// NETWORK 7: Update the step number
// Store updated step value
intSuspendStep := _intStep;
END_METHOD

(* Unpauses the device then returns TRUE. *)
METHOD M52_Unsuspend : BOOL
VAR CONSTANT
	_udintERROR_CODE: UDINT := E_DeviceControllerError.ResetError;
	_strERROR_MSG: T_MaxString := 'Error while trying to reset device!';
	_intFINAL_STEP : INT := 1000;
	_intERROR_STEP : INT := 2000;
	_strSTART_MSG: T_MaxString := 'Unsuspending device';
	_strFINISH_MSG: T_MaxString := 'Device unsuspended';
END_VAR
VAR
	_bStepComplete: BOOL;
	_intStep: INT;
END_VAR
VAR_INST // added by the converter: edge detectors and wires of the graphical bodies
    _w1, _w2, _w3, _w4, _w5, _w6, _w7 : BOOL;
END_VAR
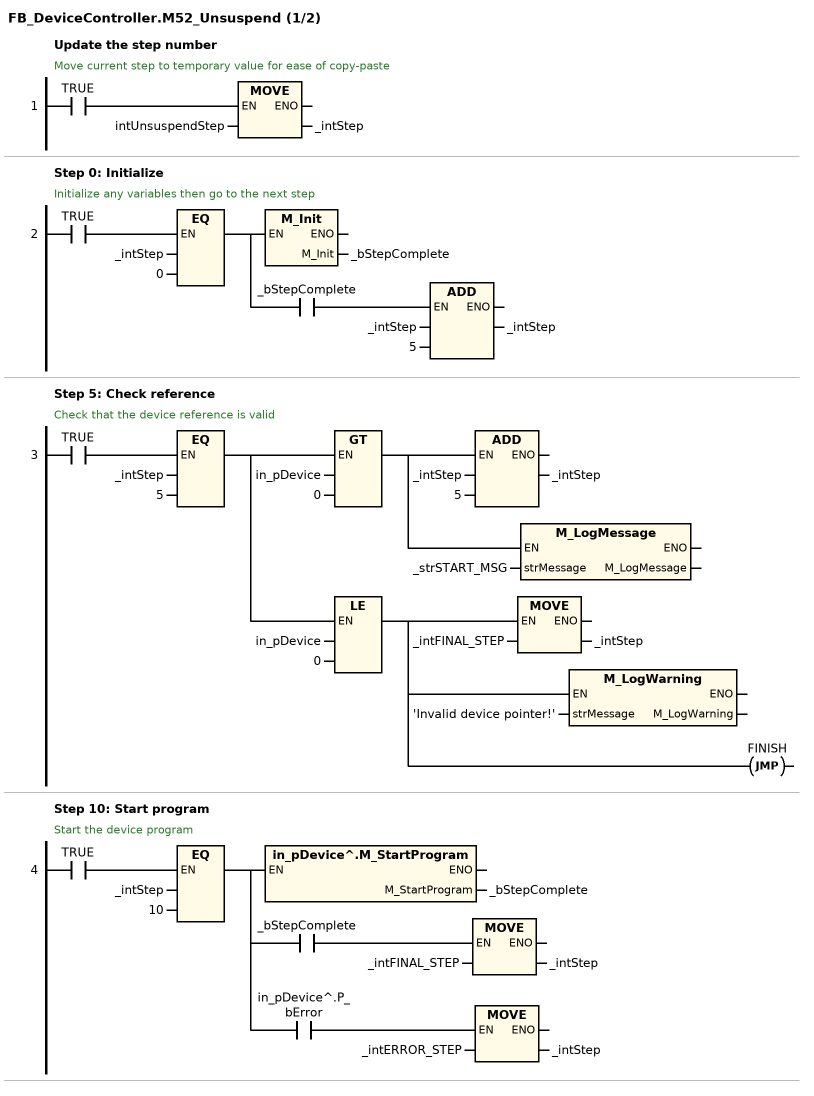
// NETWORK 1: Update the step number
// Move current step to temporary value for ease of copy-paste
_intStep := intUnsuspendStep;

// NETWORK 2: Step 0: Initialize
// Initialize any variables then go to the next step
_w1 := _intStep = 0;
IF _w1 THEN _bStepComplete := M_Init(); END_IF
IF _w1 AND _bStepComplete THEN _intStep := _intStep + 5; END_IF

// NETWORK 3: Step 5: Check reference
// Check that the device reference is valid
_w2 := _intStep = 5;
_w3 := _w2 AND in_pDevice > 0;
IF _w3 THEN _intStep := _intStep + 5; END_IF
IF _w3 THEN M_LogMessage(strMessage := _strSTART_MSG); END_IF
_w4 := _w2 AND in_pDevice <= 0;
IF _w4 THEN _intStep := _intFINAL_STEP; END_IF
IF _w4 THEN M_LogWarning(strMessage := 'Invalid device pointer!'); END_IF
IF _w4 THEN JMP FINISH; END_IF

// NETWORK 4: Step 10: Start program
// Start the device program
_w5 := _intStep = 10;
IF _w5 THEN _bStepComplete := in_pDevice^.M_StartProgram(); END_IF
IF _w5 AND _bStepComplete THEN _intStep := _intFINAL_STEP; END_IF
IF _w5 AND in_pDevice^.P_bError THEN _intStep := _intERROR_STEP; END_IF

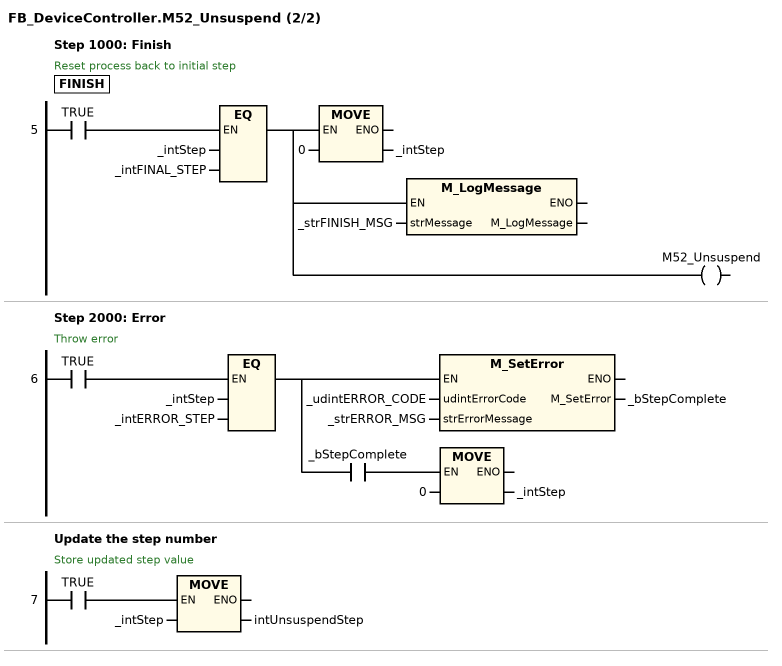
// NETWORK 5: Step 1000: Finish
// Reset process back to initial step
FINISH:
_w6 := _intStep = _intFINAL_STEP;
IF _w6 THEN _intStep := 0; END_IF
IF _w6 THEN M_LogMessage(strMessage := _strFINISH_MSG); END_IF
M52_Unsuspend := _w6;

// NETWORK 6: Step 2000: Error
// Throw error
_w7 := _intStep = _intERROR_STEP;
IF _w7 THEN
    _bStepComplete := M_SetError(udintErrorCode := _udintERROR_CODE, strErrorMessage := _strERROR_MSG);
END_IF
IF _w7 AND _bStepComplete THEN _intStep := 0; END_IF

// NETWORK 7: Update the step number
// Store updated step value
intUnsuspendStep := _intStep;
END_METHOD

END_FUNCTION_BLOCK

// Concrete/Machines/FB_SimpleMachine
(*
	Simple machine that extends and adds buttons to FB_Machine.
	If overriding any of the waiting states (including execute),
	make sure to call the SUPER^ state method to ensure the buttons
	work properly.
*)
{attribute 'hide_all_locals'}
FUNCTION_BLOCK FB_SimpleMachine EXTENDS FB_Machine IMPLEMENTS I_SimpleWaitingStatesOnly
VAR_INPUT
	(* Immediately abort all stations from whatever state they are in and
		go to the Aborted state. *)
	in_bAbortBtn : BOOL;
	(* Immediately stop all stations from whatever state they are in and
		go to the Stopped state. *)
	in_bStopBtn : BOOL;
	(* Clear all stations from the Aborted state and go to the Stopped state. *)
	in_bClearBtn : BOOL;
	(* Reset all stations from the Stopped state and go to the Idle state. *)
	in_bResetBtn : BOOL;
	(* Start all stations from the Idle state and go to the Execute state. *)
	in_bStartBtn : BOOL;
	(* Hold all stations from the Execute state and go to the Held state. *)
	in_bHoldBtn : BOOL;
	(* Unhold all stations from the Held state and go to the Execute state. *)
	in_bUnholdBtn : BOOL;
	(* Suspend all stations from the Execute state and go to the Held Suspended. *)
	in_bSuspendBtn : BOOL;
	(* Unsuspend all stations from the Suspended state and go to the Execute state. *)
	in_bUnsuspendBtn : BOOL;
	(* Complete all stations from the Execute state and go to the Completed state. *)
	in_bCompleteBtn : BOOL;
	(* Return all stations from the Completed state and go to the Idle state. *)
	in_bReturnBtn : BOOL;
END_VAR
VAR_OUTPUT
END_VAR
VAR
	// Abort
	smac_bStationError: BOOL;
	smac_fbAbortTrig: R_TRIG;
	smac_bAbortTrig: BOOL;
	smac_bAborting: BOOL;
	smac_bAborted: BOOL;

	// Stop
	smac_fbStopTrig: R_TRIG;
	smac_bStopTrig: BOOL;
	smac_bStopping: BOOL;
	smac_bStopped: BOOL;
	
	// Clear
	smac_fbClearTrig: R_TRIG;
	smac_bClearTrig: BOOL;
	smac_bClearing: BOOL;
	smac_bCleared: BOOL;
	
	// Reset
	smac_fbResetTrig: R_TRIG;
	smac_bResetTrig: BOOL;
	smac_bResetting: BOOL;
	smac_bReset: BOOL;
	
	// Start
	smac_fbStartTrig: R_TRIG;
	smac_bStartTrig: BOOL;
	smac_bStarting: BOOL;
	smac_bStarted: BOOL;
	
	// Complete
	smac_fbCompleteTrig: R_TRIG;
	smac_bCompleteTrig: BOOL;
	smac_bCompleting: BOOL;
	smac_bCompleted: BOOL;
	
	// Return
	smac_fbReturnTrig: R_TRIG;
	smac_bReturnTrig: BOOL;
	
	// Hold
	smac_fbHoldTrig: R_TRIG;
	smac_bHoldTrig: BOOL;
	smac_bHolding: BOOL;
	smac_bHeld: BOOL;
	
	// Suspend
	smac_fbSuspendTrig: R_TRIG;
	smac_bSuspendTrig: BOOL;
	smac_bSuspending: BOOL;
	smac_bSuspended: BOOL;
	
	// Unhold
	smac_fbUnholdTrig: R_TRIG;
	smac_bUnholdTrig: BOOL;
	smac_bUnholding: BOOL;
	smac_bUnheld: BOOL;
	
	// Unsuspend
	smac_fbUnsuspendTrig: R_TRIG;
	smac_bUnsuspendTrig: BOOL;
	smac_bUnsuspending: BOOL;
	smac_bUnsuspended: BOOL;
	
	// Reset variables
	smac_bResetVariables: BOOL;
END_VAR
VAR // added by the converter: edge detectors and wires of the graphical bodies
    _w1, _w2, _w3, _w4, _w5, _w6, _w7, _w8, _w9, _w10, _w11, _w12, _w13 : BOOL;
END_VAR

THIS^.A_RunSimpleMachine();

ACTION A_Buttons:
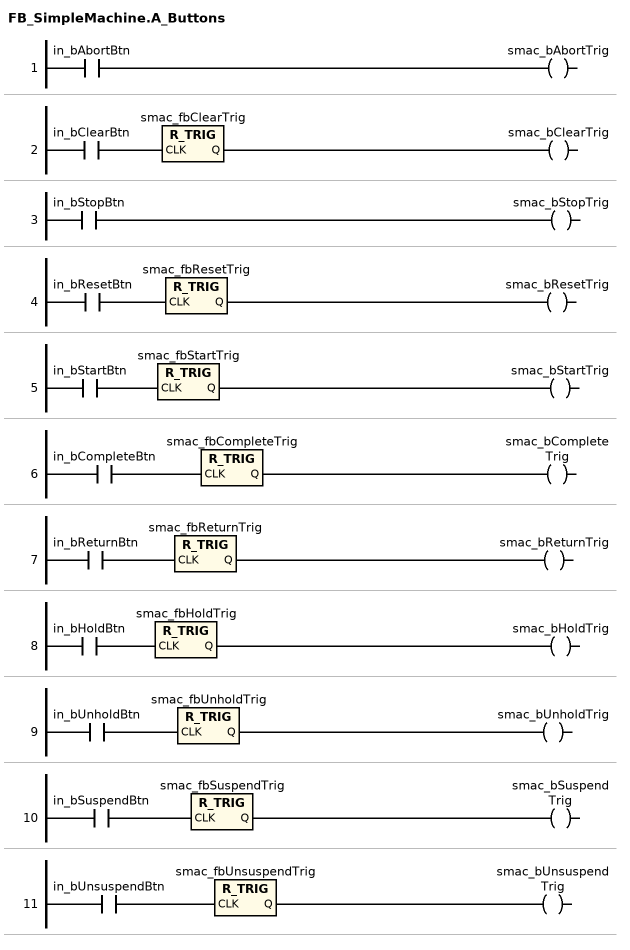
// NETWORK 1
smac_bAbortTrig := in_bAbortBtn;

// NETWORK 2
smac_fbClearTrig(CLK := in_bClearBtn); // R_TRIG
smac_bClearTrig := smac_fbClearTrig.Q;

// NETWORK 3
smac_bStopTrig := in_bStopBtn;

// NETWORK 4
smac_fbResetTrig(CLK := in_bResetBtn); // R_TRIG
smac_bResetTrig := smac_fbResetTrig.Q;

// NETWORK 5
smac_fbStartTrig(CLK := in_bStartBtn); // R_TRIG
smac_bStartTrig := smac_fbStartTrig.Q;

// NETWORK 6
smac_fbCompleteTrig(CLK := in_bCompleteBtn); // R_TRIG
smac_bCompleteTrig := smac_fbCompleteTrig.Q;

// NETWORK 7
smac_fbReturnTrig(CLK := in_bReturnBtn); // R_TRIG
smac_bReturnTrig := smac_fbReturnTrig.Q;

// NETWORK 8
smac_fbHoldTrig(CLK := in_bHoldBtn); // R_TRIG
smac_bHoldTrig := smac_fbHoldTrig.Q;

// NETWORK 9
smac_fbUnholdTrig(CLK := in_bUnholdBtn); // R_TRIG
smac_bUnholdTrig := smac_fbUnholdTrig.Q;

// NETWORK 10
smac_fbSuspendTrig(CLK := in_bSuspendBtn); // R_TRIG
smac_bSuspendTrig := smac_fbSuspendTrig.Q;

// NETWORK 11
smac_fbUnsuspendTrig(CLK := in_bUnsuspendBtn); // R_TRIG
smac_bUnsuspendTrig := smac_fbUnsuspendTrig.Q;
END_ACTION

ACTION A_RunSimpleMachine:
THIS^.A_StateControl();
THIS^.A_Buttons();
THIS^.A_StateMachine();
END_ACTION

ACTION A_StateControl:
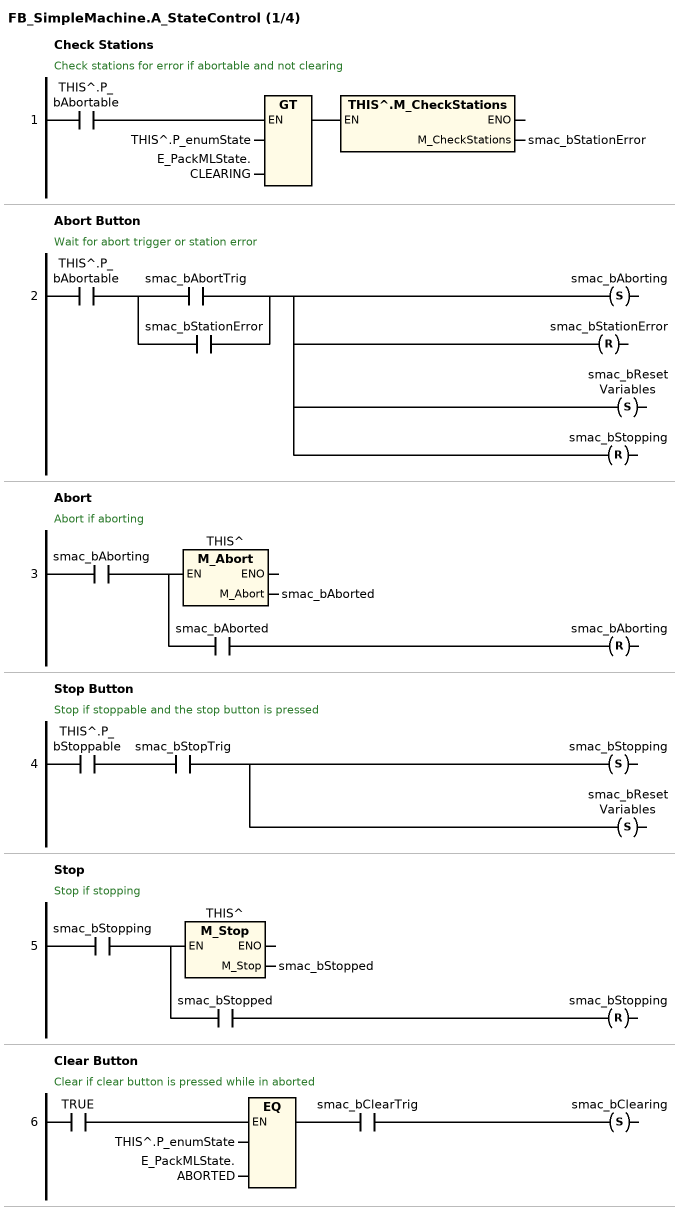
// NETWORK 1: Check Stations
// Check stations for error if abortable and not clearing
IF THIS^.P_bAbortable AND THIS^.P_enumState > E_PackMLState.CLEARING THEN
    smac_bStationError := THIS^.M_CheckStations();
END_IF

// NETWORK 2: Abort Button
// Wait for abort trigger or station error
_w1 := THIS^.P_bAbortable AND (smac_bAbortTrig OR smac_bStationError);
smac_bAborting S= _w1;
smac_bStationError R= _w1;
smac_bResetVariables S= _w1;
smac_bStopping R= _w1;

// NETWORK 3: Abort
// Abort if aborting
_w2 := smac_bAborting;
IF _w2 THEN THIS^.M_Abort(M_Abort => smac_bAborted); END_IF
smac_bAborting R= _w2 AND smac_bAborted;

// NETWORK 4: Stop Button
// Stop if stoppable and the stop button is pressed
_w3 := THIS^.P_bStoppable AND smac_bStopTrig;
smac_bStopping S= _w3;
smac_bResetVariables S= _w3;

// NETWORK 5: Stop
// Stop if stopping
_w4 := smac_bStopping;
IF _w4 THEN THIS^.M_Stop(M_Stop => smac_bStopped); END_IF
smac_bStopping R= _w4 AND smac_bStopped;

// NETWORK 6: Clear Button
// Clear if clear button is pressed while in aborted
smac_bClearing S= THIS^.P_enumState = E_PackMLState.ABORTED AND smac_bClearTrig;

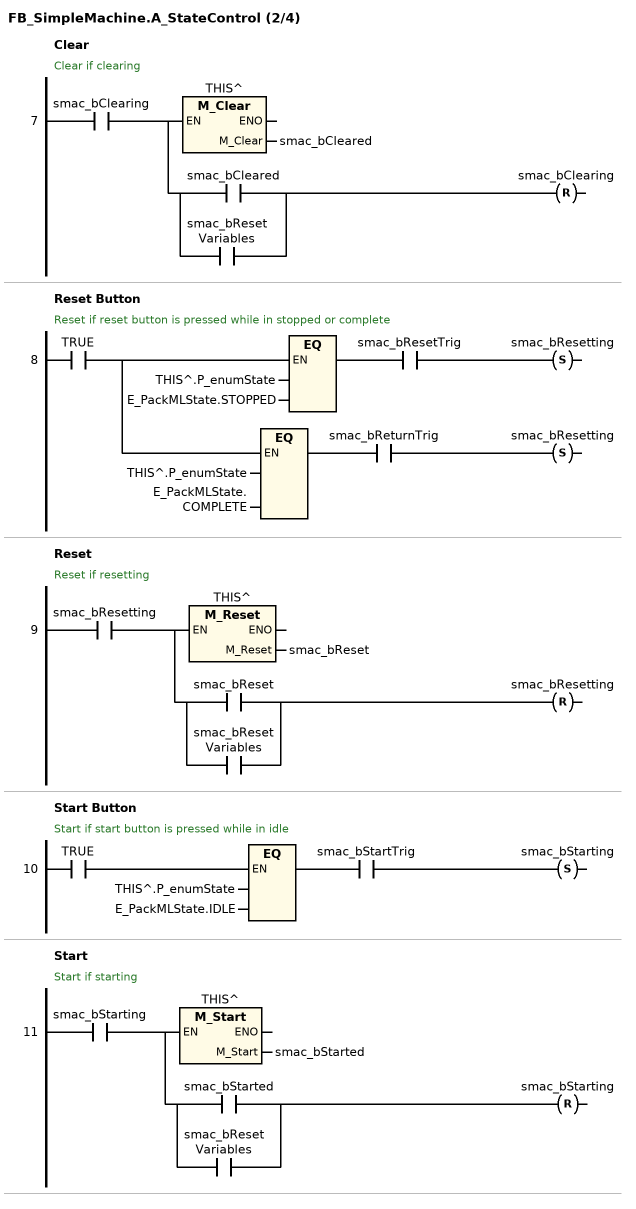
// NETWORK 7: Clear
// Clear if clearing
_w5 := smac_bClearing;
IF _w5 THEN THIS^.M_Clear(M_Clear => smac_bCleared); END_IF
smac_bClearing R= _w5 AND (smac_bCleared OR smac_bResetVariables);

// NETWORK 8: Reset Button
// Reset if reset button is pressed while in stopped or complete
smac_bResetting S= THIS^.P_enumState = E_PackMLState.STOPPED AND smac_bResetTrig;
smac_bResetting S= THIS^.P_enumState = E_PackMLState.COMPLETE AND smac_bReturnTrig;

// NETWORK 9: Reset
// Reset if resetting
_w6 := smac_bResetting;
IF _w6 THEN THIS^.M_Reset(M_Reset => smac_bReset); END_IF
smac_bResetting R= _w6 AND (smac_bReset OR smac_bResetVariables);

// NETWORK 10: Start Button
// Start if start button is pressed while in idle
smac_bStarting S= THIS^.P_enumState = E_PackMLState.IDLE AND smac_bStartTrig;

// NETWORK 11: Start
// Start if starting
_w7 := smac_bStarting;
IF _w7 THEN THIS^.M_Start(M_Start => smac_bStarted); END_IF
smac_bStarting R= _w7 AND (smac_bStarted OR smac_bResetVariables);

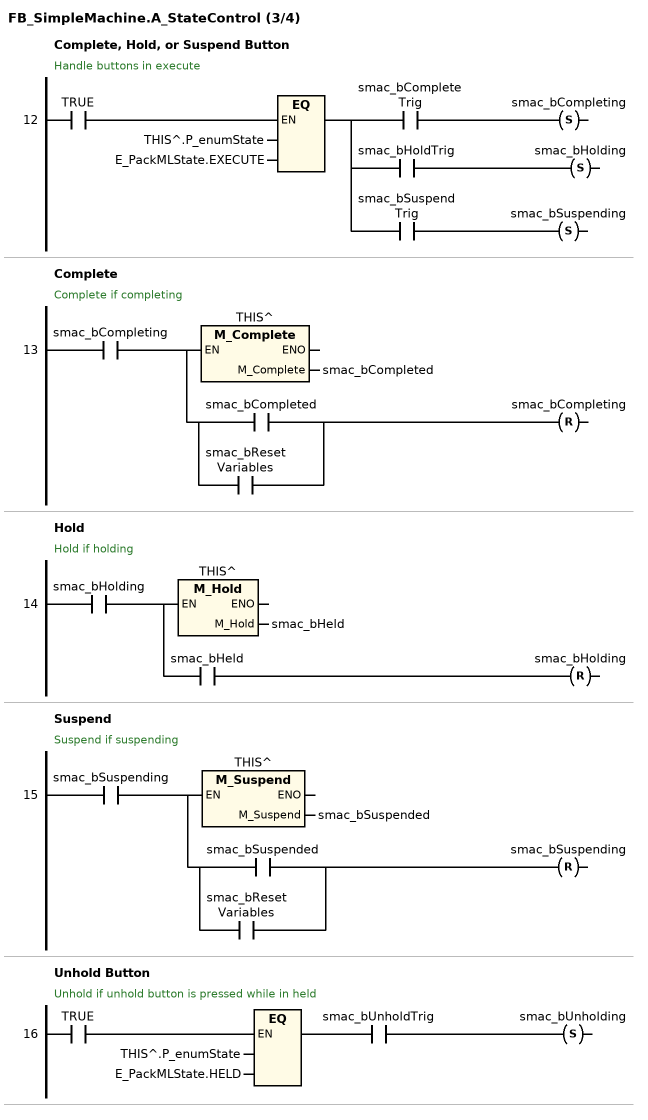
// NETWORK 12: Complete, Hold, or Suspend Button
// Handle buttons in execute
_w8 := THIS^.P_enumState = E_PackMLState.EXECUTE;
smac_bCompleting S= _w8 AND smac_bCompleteTrig;
smac_bHolding S= _w8 AND smac_bHoldTrig;
smac_bSuspending S= _w8 AND smac_bSuspendTrig;

// NETWORK 13: Complete
// Complete if completing
_w9 := smac_bCompleting;
IF _w9 THEN THIS^.M_Complete(M_Complete => smac_bCompleted); END_IF
smac_bCompleting R= _w9 AND (smac_bCompleted OR smac_bResetVariables);

// NETWORK 14: Hold
// Hold if holding
_w10 := smac_bHolding;
IF _w10 THEN THIS^.M_Hold(M_Hold => smac_bHeld); END_IF
smac_bHolding R= _w10 AND smac_bHeld;

// NETWORK 15: Suspend
// Suspend if suspending
_w11 := smac_bSuspending;
IF _w11 THEN THIS^.M_Suspend(M_Suspend => smac_bSuspended); END_IF
smac_bSuspending R= _w11 AND (smac_bSuspended OR smac_bResetVariables);

// NETWORK 16: Unhold Button
// Unhold if unhold button is pressed while in held
smac_bUnholding S= THIS^.P_enumState = E_PackMLState.HELD AND smac_bUnholdTrig;

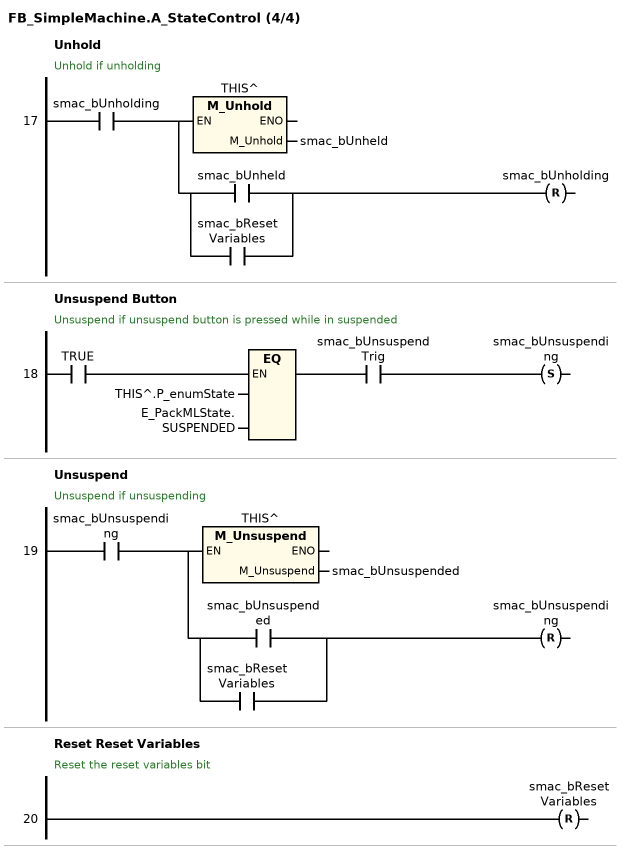
// NETWORK 17: Unhold
// Unhold if unholding
_w12 := smac_bUnholding;
IF _w12 THEN THIS^.M_Unhold(M_Unhold => smac_bUnheld); END_IF
smac_bUnholding R= _w12 AND (smac_bUnheld OR smac_bResetVariables);

// NETWORK 18: Unsuspend Button
// Unsuspend if unsuspend button is pressed while in suspended
smac_bUnsuspending S= THIS^.P_enumState = E_PackMLState.SUSPENDED AND smac_bUnsuspendTrig;

// NETWORK 19: Unsuspend
// Unsuspend if unsuspending
_w13 := smac_bUnsuspending;
IF _w13 THEN THIS^.M_Unsuspend(M_Unsuspend => smac_bUnsuspended); END_IF
smac_bUnsuspending R= _w13 AND (smac_bUnsuspended OR smac_bResetVariables);

// NETWORK 20: Reset Reset Variables
// Reset the reset variables bit
smac_bResetVariables R= TRUE;
END_ACTION

END_FUNCTION_BLOCK

// Concrete/Machines/FB_StandardMachine
FUNCTION_BLOCK FB_StandardMachine EXTENDS FB_Machine
	IMPLEMENTS I_UserControls
VAR_INPUT
	(* Struct of state change commands. *)
	in_stCommands: ST_PackMLStateCommands;
	(* Array of user prompts. *)
	in_arrUserPrompts: ARRAY[1..GVL_Constants.intMAX_USER_PROMPTS] OF ST_Prompt;
	(* User retry signal for an exception state. *)
	in_bUserRetry: BOOL;
	(* User stop machine signal for an exception state. *)
	in_bUserAbort: BOOL;
	(* Array of resync requests for each station. *)
	in_arrResyncRequest: ARRAY[1..GVL_Constants.uintMAX_MACHINE_STATION_COUNT] OF BOOL;
END_VAR
VAR_OUTPUT
	(* ID of the current user prompt. *)
	out_udintUserPromptCode: UDINT;
	(* Default message of the current user prompt. *)
	out_strUserPromptMessage: T_MaxString;
	(* TRUE if a station is not synchronized. *)
	out_arrStationDesynched: ARRAY[1..GVL_Constants.uintMAX_MACHINE_STATION_COUNT] OF BOOL;
END_VAR
VAR
	// Abort
	smac_bStationError: BOOL;
	smac_fbAbortTrig: R_TRIG;
	smac_bAbortTrig: BOOL;
	smac_bAborting: BOOL;
	smac_bAborted: BOOL;

	// Stop
	smac_fbStopTrig: R_TRIG;
	smac_bStopTrig: BOOL;
	smac_bStopping: BOOL;
	smac_bStopped: BOOL;
	
	// Clear
	smac_fbClearTrig: R_TRIG;
	smac_bClearTrig: BOOL;
	smac_bClearing: BOOL;
	smac_bCleared: BOOL;
	
	// Reset
	smac_fbResetTrig: R_TRIG;
	smac_bResetTrig: BOOL;
	smac_bResetting: BOOL;
	smac_bReset: BOOL;
	
	// Start
	smac_fbStartTrig: R_TRIG;
	smac_bStartTrig: BOOL;
	smac_bStarting: BOOL;
	smac_bStarted: BOOL;
	
	// Complete
	smac_fbCompleteTrig: R_TRIG;
	smac_bCompleteTrig: BOOL;
	smac_bCompleting: BOOL;
	smac_bCompleted: BOOL;
	
	// Return
	smac_fbReturnTrig: R_TRIG;
	smac_bReturnTrig: BOOL;
	
	// Hold
	smac_fbHoldTrig: R_TRIG;
	smac_bHoldTrig: BOOL;
	smac_bHolding: BOOL;
	smac_bHeld: BOOL;
	
	// Suspend
	smac_fbSuspendTrig: R_TRIG;
	smac_bSuspendTrig: BOOL;
	smac_bSuspending: BOOL;
	smac_bSuspended: BOOL;
	
	// Unhold
	smac_fbUnholdTrig: R_TRIG;
	smac_bUnholdTrig: BOOL;
	smac_bUnholding: BOOL;
	smac_bUnheld: BOOL;
	
	// Unsuspend
	smac_fbUnsuspendTrig: R_TRIG;
	smac_bUnsuspendTrig: BOOL;
	smac_bUnsuspending: BOOL;
	smac_bUnsuspended: BOOL;
	
	// Reset variables
	smac_bResetVariables: BOOL;
	
	stdmac_intIndex: INT;
	stdmac_enumStationState: E_PackMLState;
	stdmac_arrResyncState: ARRAY[1..GVL_Constants.uintMAX_MACHINE_STATION_COUNT] OF INT;
	stdmac_intResyncState: INT;
	stdmac_bResyncRequest: BOOL;
	stdmac_enumStateRequest: E_PackMLSTate;
	stdmac_enumMachineState: E_PackMLState;
END_VAR
VAR // added by the converter: edge detectors and wires of the graphical bodies
    _w1, _w2, _w3, _w4, _w5, _w6, _w7, _w8, _w9, _w10, _w11, _w12, _w13 : BOOL;
END_VAR

(* Clears the user prompt outputs. *)
METHOD M_ClearUserPrompt : BOOL
VAR_INPUT
END_VAR
out_strUserPromptMessage := '';
out_udintUserPromptCode := 0;
M_ClearUserPrompt := TRUE;
END_METHOD

(* Sets user prompt based on given code, and awaits user input. *)
METHOD M_HandleException : BOOL
VAR_INPUT
	(* Prompt code for the exception message. *)
	_in_udintPromptCode: UDINT;
	(* Error code to set in case user aborts. *)
	_in_udintErrorCode: UDINT;
END_VAR
VAR_OUTPUT
END_VAR
M_HandleException := FALSE;
THIS^.M_SetUserPrompt(_in_udintPromptCode);
IF in_bUserRetry THEN
	THIS^.M_ClearUserPrompt();
	M_HandleException := TRUE;
ELSIF in_bUserAbort THEN
	THIS^.M_SetError(_in_udintErrorCode, 'User chose to abort after an exception.');
END_IF
END_METHOD

(* Sets out_strUserPromptCode and out_strUserPromptMessage based on
	the given user prompt code. *)
METHOD M_SetUserPrompt : BOOL
VAR_INPUT
	(* Prompt code to use for this user prompt. *)
	_in_udintCode: UDINT;
END_VAR

VAR
	_strMessage: T_MaxString;
	_intIndex: INT;
END_VAR
FOR _intIndex := 1 TO GVL_Constants.intMAX_USER_PROMPTS DO
	IF in_arrUserPrompts[_intIndex].udintCode = _in_udintCode THEN
		_strMessage := in_arrUserPrompts[_intIndex].strMessage;
		EXIT;
	END_IF
END_FOR
IF out_udintUserPromptCode <> _in_udintCode THEN
	IF LEN(_strMessage) > 0 THEN
		THIS^.M_LogMessage(_strMessage);
	ELSE
		THIS^.M_LogWarning('Prompt message not found!');
	END_IF
END_IF
out_strUserPromptMessage := _strMessage;
out_udintUserPromptCode := _in_udintCode;
M_SetUserPrompt := TRUE;
END_METHOD

ACTION A_Buttons:
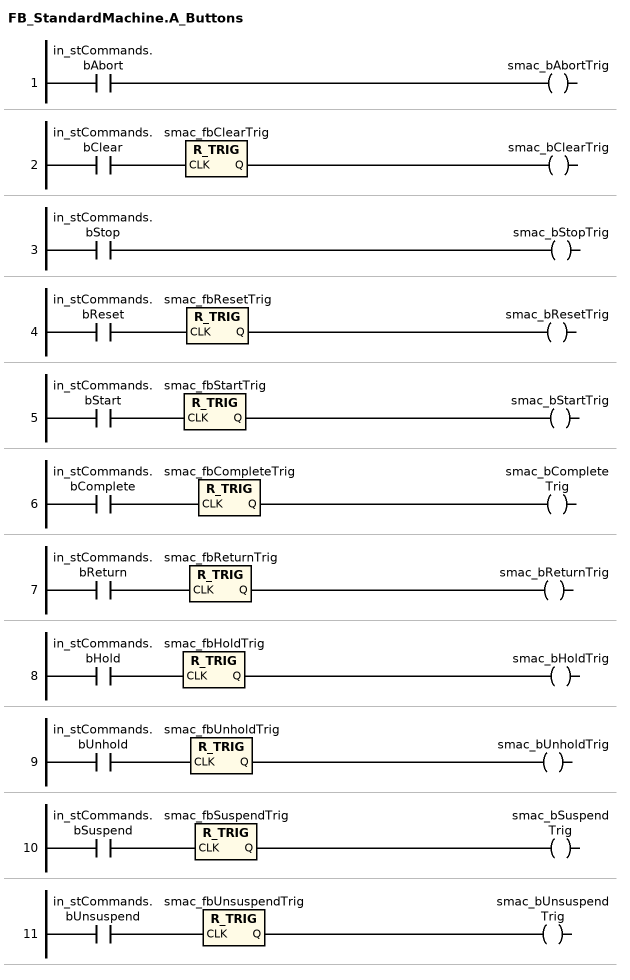
// NETWORK 1
smac_bAbortTrig := in_stCommands.bAbort;

// NETWORK 2
smac_fbClearTrig(CLK := in_stCommands.bClear); // R_TRIG
smac_bClearTrig := smac_fbClearTrig.Q;

// NETWORK 3
smac_bStopTrig := in_stCommands.bStop;

// NETWORK 4
smac_fbResetTrig(CLK := in_stCommands.bReset); // R_TRIG
smac_bResetTrig := smac_fbResetTrig.Q;

// NETWORK 5
smac_fbStartTrig(CLK := in_stCommands.bStart); // R_TRIG
smac_bStartTrig := smac_fbStartTrig.Q;

// NETWORK 6
smac_fbCompleteTrig(CLK := in_stCommands.bComplete); // R_TRIG
smac_bCompleteTrig := smac_fbCompleteTrig.Q;

// NETWORK 7
smac_fbReturnTrig(CLK := in_stCommands.bReturn); // R_TRIG
smac_bReturnTrig := smac_fbReturnTrig.Q;

// NETWORK 8
smac_fbHoldTrig(CLK := in_stCommands.bHold); // R_TRIG
smac_bHoldTrig := smac_fbHoldTrig.Q;

// NETWORK 9
smac_fbUnholdTrig(CLK := in_stCommands.bUnhold); // R_TRIG
smac_bUnholdTrig := smac_fbUnholdTrig.Q;

// NETWORK 10
smac_fbSuspendTrig(CLK := in_stCommands.bSuspend); // R_TRIG
smac_bSuspendTrig := smac_fbSuspendTrig.Q;

// NETWORK 11
smac_fbUnsuspendTrig(CLK := in_stCommands.bUnsuspend); // R_TRIG
smac_bUnsuspendTrig := smac_fbUnsuspendTrig.Q;
END_ACTION

ACTION A_Resync:
FOR stdmac_intIndex := 1 TO UINT_TO_INT(GVL_Constants.uintMAX_MACHINE_STATION_COUNT) DO
	// Exit if pointer is not assigned
	IF mac_arrStations[stdmac_intIndex] = 0 THEN
		CONTINUE;
	END_IF
	
	// Resync state machine
	stdmac_intResyncState := stdmac_arrResyncState[stdmac_intIndex];
	stdmac_bResyncRequest := in_arrResyncRequest[stdmac_intIndex];
	CASE stdmac_intResyncState OF
		0:	// Wait for request reset
			IF NOT stdmac_bResyncRequest THEN
				stdmac_intResyncState := 10;
			END_IF
			
		10: // Wait for request when station is desynched
			IF out_arrStationDesynched[stdmac_intIndex] AND stdmac_bResyncRequest THEN
				stdmac_intResyncState := 20;
			END_IF
			
		20: // Resync the station
			stdmac_enumStateRequest := THIS^.P_enumState;
			mac_arrStations[stdmac_intIndex]^.M_MoveToState(stdmac_enumStateRequest);
			IF NOT out_arrStationDesynched[stdmac_intIndex] THEN
				stdmac_intResyncState := 0;
			END_IF
	END_CASE
	stdmac_arrResyncState[stdmac_intIndex] := stdmac_intResyncState;
END_FOR
END_ACTION

ACTION A_RunStandardMachine:
A_StateMachine();
A_Buttons();
A_StateControl();
A_TrackSync();
A_Resync();
END_ACTION

ACTION A_StateControl:
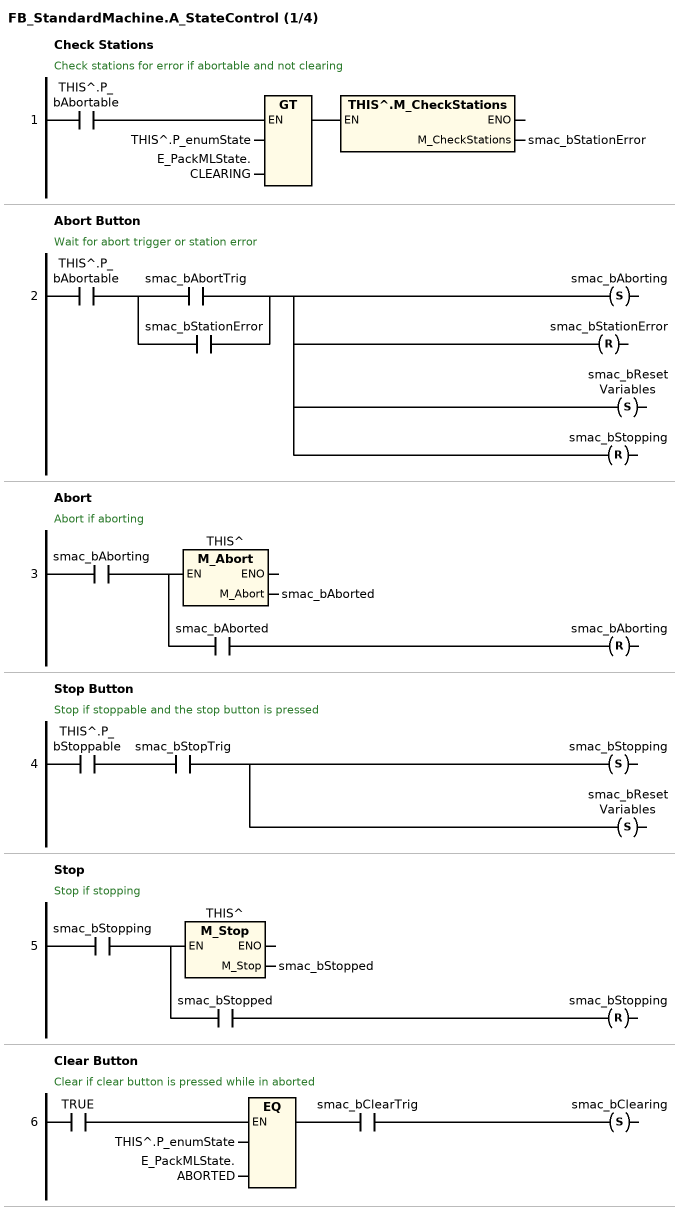
// NETWORK 1: Check Stations
// Check stations for error if abortable and not clearing
IF THIS^.P_bAbortable AND THIS^.P_enumState > E_PackMLState.CLEARING THEN
    smac_bStationError := THIS^.M_CheckStations();
END_IF

// NETWORK 2: Abort Button
// Wait for abort trigger or station error
_w1 := THIS^.P_bAbortable AND (smac_bAbortTrig OR smac_bStationError);
smac_bAborting S= _w1;
smac_bStationError R= _w1;
smac_bResetVariables S= _w1;
smac_bStopping R= _w1;

// NETWORK 3: Abort
// Abort if aborting
_w2 := smac_bAborting;
IF _w2 THEN THIS^.M_Abort(M_Abort => smac_bAborted); END_IF
smac_bAborting R= _w2 AND smac_bAborted;

// NETWORK 4: Stop Button
// Stop if stoppable and the stop button is pressed
_w3 := THIS^.P_bStoppable AND smac_bStopTrig;
smac_bStopping S= _w3;
smac_bResetVariables S= _w3;

// NETWORK 5: Stop
// Stop if stopping
_w4 := smac_bStopping;
IF _w4 THEN THIS^.M_Stop(M_Stop => smac_bStopped); END_IF
smac_bStopping R= _w4 AND smac_bStopped;

// NETWORK 6: Clear Button
// Clear if clear button is pressed while in aborted
smac_bClearing S= THIS^.P_enumState = E_PackMLState.ABORTED AND smac_bClearTrig;

